Universal Robots PolyScope program: Cooperation_QualityInspection.urp

Program Cooperation_QualityInspection (installation=Cooperation_QualityInspection directory=/home/cobot/ursim-5.11.5.1010327/programs createdIn=5.11.5.1010327 lastSavedIn=5.11.5.1010327 robotSerialNumber=20195599999)
Calibrated DH parameters: a=[0, -0.425, -0.3922, 0, 0, 0]; d=[0.1625, 0, 0, 0.1333, 0.0997, 0.0996]; alpha=[1.570796, 0, 0, 1.570796, -1.570796, 0]; deltaTheta=[0, 0, 0, 0, 0, 0]
Robot Program (runOnlyOnce=false)
  Wait DigitalInput pin=ib64; digitalValue=1
  Switch expression=ii24_step
    Case (caseValue=1)
      'Move to Home position'
      SafeHome (positionOptionType=SPEED_AND_ACCELERATION speed=1.047198 acceleration=1.396263 nextMotionTime=2)
    Case (caseValue=2)
      MoveL speed 250 mm/s, acceleration 1200 mm/s^2 (useActiveTCP=true) feature=Base
        Waypoint Waypoint (Variable): variable(featureName=WaitPos)
      'Read inspectionPos'
      inspectionPos := p[if24_x,if25_y,if26_z,if27_rx,if28_ry,if29_rz]
      'Move: inspectionPos'
      Switch expression=GP_int_in[25]
        Case (caseValue=1)
          MoveL speed 250 mm/s, acceleration 1200 mm/s^2 (useActiveTCP=true) feature=BackLeftBot_1
            Waypoint Waypoint (Variable): variable=inspectionPos
        Case (caseValue=2)
          MoveL speed 250 mm/s, acceleration 1200 mm/s^2 (useActiveTCP=true) feature=BackLeftBot_2
            Waypoint Waypoint (Variable): variable=inspectionPos
        Case (caseValue=3)
          MoveL speed 250 mm/s, acceleration 1200 mm/s^2 (useActiveTCP=true) feature=BackLeftTop_1
            Waypoint Waypoint (Variable): variable=inspectionPos
        Case (caseValue=4)
          MoveL speed 250 mm/s, acceleration 1200 mm/s^2 (useActiveTCP=true) feature=BackLeftTop_2
            Waypoint Waypoint (Variable): variable=inspectionPos
        Case (caseValue=5)
          MoveL speed 250 mm/s, acceleration 1200 mm/s^2 (useActiveTCP=true) feature=BackRightBot_1
            Waypoint Waypoint (Variable): variable=inspectionPos
        Case (caseValue=6)
          MoveL speed 250 mm/s, acceleration 1200 mm/s^2 (useActiveTCP=true) feature=BackRightBot_2
            Waypoint Waypoint (Variable): variable=inspectionPos
        Case (caseValue=7)
          MoveL speed 250 mm/s, acceleration 1200 mm/s^2 (useActiveTCP=true) feature=BackRightTop_1
            Waypoint Waypoint (Variable): variable=inspectionPos
        Case (caseValue=8)
          MoveL speed 250 mm/s, acceleration 1200 mm/s^2 (useActiveTCP=true) feature=BackRightTop_2
            Waypoint Waypoint (Variable): variable=inspectionPos
    Case (caseValue=2147483647)
      'Do nothing (just handshake)'
  Set DigitalOutput pin=ob64; digitalValue=1
  Wait DigitalInput pin=ib64; digitalValue=0
  Set DigitalOutput pin=ob64; digitalValue=0
